FUNCTION_BLOCK Heating_State_Enabled EXTENDS Heating_State
VAR_INPUT
END_VAR
VAR_OUTPUT
END_VAR
VAR
END_VAR

METHOD OnExecute
VAR
	_iRoomArg		: I_Arg;
END_VAR
IF _ctx.hmi.bButton THEN
	_ctx.hmi.bButton := FALSE;
	_ctx.state.iMgr.Request(_ctx.state.iDisable);
	
ELSIF _ctx.io.in.rBoilerTemp < _ctx.hmi.rMinTemperature THEN
	_ctx.state.iMgr.Request(_ctx.state.iHeatup);
	
ELSIF IsOk(_ctx.priv.iQueue.Pop(iArg => _iRoomArg)) THEN
	IF IsOk(ArgAsIRoom(_iRoomArg, iDest => _ctx.priv.iActiveRoom)) THEN
		_ctx.state.iMgr.Request(_ctx.state.iPump);
	ELSE
		_ctx.hmi.sErrorText := 'Room Queue - Incorrect iRoomArg!';
	END_IF
END_IF

IF NOT _ctx.io.out.bPump AND _ctx.priv.nPassiveRooms <> 0 THEN
	_ctx.io.out.bPump := TRUE;
	_ctx.hmi.sStatusText := 'Heating enabled: Circulating...';
	
ELSIF _ctx.io.out.bPump AND _ctx.priv.nPassiveRooms <> 0 THEN
	_ctx.io.out.bPump := FALSE;
	_ctx.hmi.sStatusText := 'Heating enabled: Waiting for requests...';
	
END_IF
END_METHOD

METHOD OnInit
_ctx.hmi.sStatusText := 'Heating enabled: Waiting for requests...';
_ctx.hmi.nStatusColor := COL.BLACK.Raw;

_ctx.hmi.sButtonText := 'Press to DISABLE!';
_ctx.hmi.nButtonColor := COL.BLACK.Raw;

_ctx.io.out.bBurner := FALSE;
_ctx.io.out.bPump := FALSE;

_ctx.priv.iOnEnable.Emit();
_ctx.priv.iOnResume.Emit();
END_METHOD

END_FUNCTION_BLOCK

(* stored: Version 1.1.0.1
   POU Heating_State_Enabled: Id {dbdd9ce5-7113-42e8-8cbb-47f12de11ae0}, SpecialFunc None
   Method OnExecute: Id {8515d0dd-e19e-4fb0-85ae-5b4ce34b6e10}
   Method OnInit: Id {ff2ff1ed-67cd-4bcc-bf07-4aeaf2a4bb97} *)
